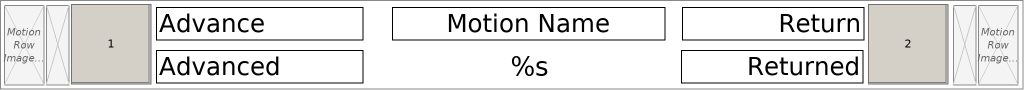
VISUALIZATION MotionRow  // 1024x90
    Button (868,4 80x80), "2", text variable: MotionRowInstanceSingle.Returned.NumberOrder, invisible if: MotionRowInstanceSingle.Returned.bHideButton, text list: 'MotionRowText', text index: MotionRowInstanceSingle.IndexLocation + 5
        tap MotionRowButtonsSingle.btnReturn
    Rectangle (682,7 182x33), "Return", colour toggle: MotionRowInstanceSingle.Returned.RequestCoil, invisible if: MotionRowInstanceSingle.Returned.bHideCoil, text list: 'MotionRowText', text index: MotionRowInstanceSingle.IndexLocation + 3
    Rectangle (392,7 273x33), "Motion Name", invisible if: MotionRowInstanceSingle.bHideName, text list: 'MotionRowText', text index: MotionRowInstanceSingle.IndexLocation + 6
    Rectangle (681,50 182x33), "Returned", colour toggle: MotionRowInstanceSingle.Returned.Depth, invisible if: MotionRowInstanceSingle.Returned.bHideDepth, text list: 'MotionRowText', text index: MotionRowInstanceSingle.IndexLocation + 4
    Rectangle (156,7 207x33), "Advance", text variable: MotionRowInstanceSingle.Advance.valCoil, colour toggle: MotionRowInstanceSingle.Advance.RequestCoil, invisible if: MotionRowInstanceSingle.Advance.bHideCoil, text list: 'MotionRowText', text index: MotionRowInstanceSingle.IndexLocation + 0
    Button (71,4 80x80), "1", invisible if: MotionRowInstanceSingle.Advance.bHideButton, text list: 'MotionRowText', text index: MotionRowInstanceSingle.IndexLocation + 2
        tap MotionRowButtonsSingle.btnAdvance
    Rectangle (393,50 273x33), "%s", text variable: MotionRowInstanceSingle.strPosn, invisible if: MotionRowInstanceSingle.bHidePosn
    Rectangle (156,50 207x33), "Advanced", colour toggle: MotionRowInstanceSingle.Advance.Depth, invisible if: MotionRowInstanceSingle.Advance.bHideDepth, text list: 'MotionRowText', text index: MotionRowInstanceSingle.IndexLocation + 1
    Image (4,5 40x80), invisible if: NOT MotionRowInstanceSingle.Advance.InterlockOK OR MotionRowInstanceSingle.Advance.bHideInterlock, image: MotionRowImages.LeftHighlight
    Image (4,5 40x80), invisible if: MotionRowInstanceSingle.Advance.InterlockOK OR MotionRowInstanceSingle.Advance.bHideInterlock, image: MotionRowImages.LeftNot
    Image (978,5 40x80), invisible if: MotionRowInstanceSingle.Returned.InterlockOK OR MotionRowInstanceSingle.Returned.bHideInterlock, image: MotionRowImages.RightNot
    Image (978,5 40x80), invisible if: NOT MotionRowInstanceSingle.Returned.InterlockOK OR MotionRowInstanceSingle.Returned.bHideInterlock, image: MotionRowImages.RightHighlight
    Image (46,5 23x80), invisible if: MotionRowInstanceSingle.Advance.Prompt OR MotionRowInstanceSingle.Advance.bHidePrompt, image: MotionRowImages.PromptNOK
    Image (953,5 23x80), invisible if: NOT MotionRowInstanceSingle.Returned.Prompt OR MotionRowInstanceSingle.Returned.bHidePrompt, image: MotionRowImages.PromptOK
    Image (953,5 23x80), invisible if: MotionRowInstanceSingle.Returned.Prompt OR MotionRowInstanceSingle.Returned.bHidePrompt, image: MotionRowImages.PromptNOK
    Image (46,5 23x80), invisible if: NOT MotionRowInstanceSingle.Advance.Prompt OR MotionRowInstanceSingle.Advance.bHidePrompt, image: MotionRowImages.PromptOK
END_VISUALIZATION

(* stored: Version 1.1.0.1, ProductVersion 3.1.4024.12
   Visu MotionRow: Id {23ea9bd1-da8d-4de5-b75e-eda7cd7af884} *)
